FUNCTION_BLOCK ModeSelect IMPLEMENTS ITF_ModeSelect
VAR
	fb_mem : STRUCT_ModeSelect;
END_VAR

(*
$$$$$$$$\                                                                   $$\       $$$$$$$$\                     $$\                                         $$\                     
$$  _____|                                                                  $$ |      $$  _____|                    \__|                                        \__|                    
$$ |   $$$$$$\   $$$$$$\  $$$$$$$\  $$\  $$\  $$\  $$$$$$\   $$$$$$\   $$$$$$$ |      $$ |      $$$$$$$\   $$$$$$\  $$\ $$$$$$$\   $$$$$$\   $$$$$$\   $$$$$$\  $$\ $$$$$$$\   $$$$$$\  
$$$$$\ \____$$\ $$  __$$\ $$  __$$\ $$ | $$ | $$ |$$  __$$\ $$  __$$\ $$  __$$ |      $$$$$\    $$  __$$\ $$  __$$\ $$ |$$  __$$\ $$  __$$\ $$  __$$\ $$  __$$\ $$ |$$  __$$\ $$  __$$\ 
$$  __|$$$$$$$ |$$ |  \__|$$ |  $$ |$$ | $$ | $$ |$$ /  $$ |$$ /  $$ |$$ /  $$ |      $$  __|   $$ |  $$ |$$ /  $$ |$$ |$$ |  $$ |$$$$$$$$ |$$$$$$$$ |$$ |  \__|$$ |$$ |  $$ |$$ /  $$ |
$$ |  $$  __$$ |$$ |      $$ |  $$ |$$ | $$ | $$ |$$ |  $$ |$$ |  $$ |$$ |  $$ |      $$ |      $$ |  $$ |$$ |  $$ |$$ |$$ |  $$ |$$   ____|$$   ____|$$ |      $$ |$$ |  $$ |$$ |  $$ |
$$ |  \$$$$$$$ |$$ |      $$ |  $$ |\$$$$$\$$$$  |\$$$$$$  |\$$$$$$  |\$$$$$$$ |      $$$$$$$$\ $$ |  $$ |\$$$$$$$ |$$ |$$ |  $$ |\$$$$$$$\ \$$$$$$$\ $$ |      $$ |$$ |  $$ |\$$$$$$$ |
\__|   \_______|\__|      \__|  \__| \_____\____/  \______/  \______/  \_______|      \________|\__|  \__| \____$$ |\__|\__|  \__| \_______| \_______|\__|      \__|\__|  \__| \____$$ |
                                                                                                          $$\   $$ |                                                          $$\   $$ |
                                                                                                          \$$$$$$  |                                                          \$$$$$$  |
                                                                                                           \______/                                                            \______/ 
*)

{warning 'add method implementation '}
METHOD Auto : BOOL
fb_mem.Auto 	:= TRUE;
fb_mem.Manueel 	:= FALSE;

RETURN(fb_mem.Auto);
END_METHOD

{warning 'add method implementation '}
METHOD Manueel : BOOL
fb_mem.Auto 	:= FALSE;
fb_mem.Manueel 	:= TRUE;

RETURN(fb_mem.Manueel);
END_METHOD

{warning 'add property implementation'}
PROPERTY Tag : STRING
GET
Tag := fb_mem.Tag;
END_GET
SET
fb_mem.Tag := Tag;
END_SET
END_PROPERTY

END_FUNCTION_BLOCK

(* stored: Version 1.1.0.1, ProductVersion 3.1.4024.12
   POU ModeSelect: Id {5ed98344-65a1-4237-8e95-92b76448fb41}, SpecialFunc None
   Method Auto: Id {d3d5499c-2109-42c6-be18-56c702aa1a2f}
   Method Manueel: Id {007bec01-c966-4e5f-bc86-f259586d9482}
   Property Tag: Id {c0961889-91d3-4152-90f8-549846efc6f0}
   Get Get: Id {e9d2bcc8-6429-4fbe-be25-dcdce6450c27}
   Set Set: Id {5bc8c772-bae3-40ba-8cda-c81304843143} *)
